# EPICS StreamDevice protocol: MotorDriverApp/Db/MotorDriver.proto
ReplyTimeout=1000;
ReadTimeout =1000;
InTerminator=CR LF;

getData {
    separator=', ';
    out "DATA?";
    in  "DATA [%f]";
}

getEnbl {
    out "DRV_ENBL?";
    in  "DRV_ENBL %i";
}

setEnbl {
    out "DRV_ENBL %i";
    in  "DRV_ENBL %i";
}
